(* IEC 61131-3 sources: CodesysTest/export/ObjectHandling/FB_CollectionHandlerInitializable.pou, 1 file *)

(* ---- InitializeAll.m.st ---- *)
(*#-#-#-#-#-#-#-#-#-#---Declaration---#-#-#-#-#-#-#-#-#-#-#-#-#*)

METHOD InitializeAll
VAR_INPUT

END_VAR
VAR
	J : UINT;
	Cast : IInitializable;
END_VAR
(*#-#-#-#-#-#-#-#-#-#---Implementation---#-#-#-#-#-#-#-#-#-#-#-#-#*)

FOR J:= 0 TO _TotalObj - 1 DO
	IF (__QUERYINTERFACE(Collection[J], Cast)) THEN
		Cast.Initialize();
	ELSE
		RETURN;
	END_IF
END_FOR
